TYPE ST_Encoder_HMI EXTENDS ST_HmiFunction :
	STRUCT
		Config			 : ST_EncoderConfig_HMI;
		ActualSpeed		 : LREAL;
		ActualPosition	 : LREAL;
		RawValueSpeed	 : INT;
		RawValuePosition : UINT;
	END_STRUCT
END_TYPE

(* stored: Version 1.1.0.1
   DUT ST_Encoder_HMI: Id {4ac4e9a7-ea1c-4e44-820b-ce9159a28136} *)
